Staubli VAL3: OnF2.pgx

program OnF2()
begin
  //
  if find(sItem,"O")!=-1
    if dOut[sIOName]==true
      dOut[sIOName]=false
    endIf
  else
    popUpMsg("对输入量无效。")
  endIf


end
